TYPE ST_MyType :
STRUCT
	bValue 	: BOOL;
	iValue	: INT := 100;
	sText	: STRING := 'Hallo Welt';
END_STRUCT
END_TYPE

(* stored: Version 1.1.0.1, ProductVersion 3.1.4024.12
   DUT ST_MyType: Id {7aaeb4d1-0f5b-4203-9ba4-0081c510af4f} *)
